PROGRAM POU_AxisClearError
VAR_INPUT
END_VAR
VAR
	fbAxis1Reset:MC_Reset;
	fbAxis2Reset:MC_Reset;
	fbAxis3Reset:MC_Reset;
	fbAxis4Reset:MC_Reset;
	fbAxis5Reset:MC_Reset;
	fbAxis6Reset:MC_Reset;
	
END_VAR

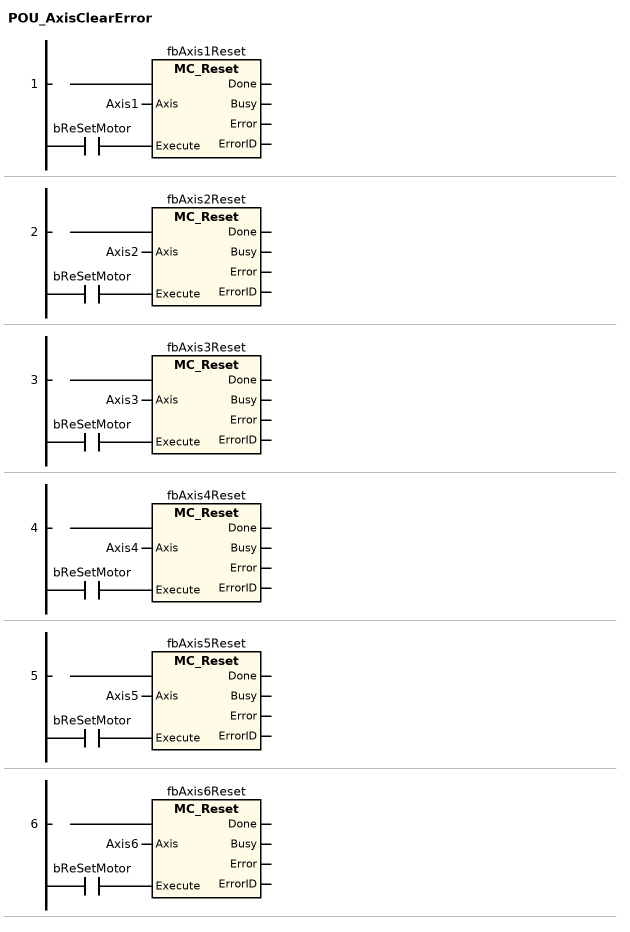
// NETWORK 1
fbAxis1Reset(Axis := Axis1, Execute := bReSetMotor); // MC_Reset

// NETWORK 2
fbAxis2Reset(Axis := Axis2, Execute := bReSetMotor); // MC_Reset

// NETWORK 3
fbAxis3Reset(Axis := Axis3, Execute := bReSetMotor); // MC_Reset

// NETWORK 4
fbAxis4Reset(Axis := Axis4, Execute := bReSetMotor); // MC_Reset

// NETWORK 5
fbAxis5Reset(Axis := Axis5, Execute := bReSetMotor); // MC_Reset

// NETWORK 6
fbAxis6Reset(Axis := Axis6, Execute := bReSetMotor); // MC_Reset

END_PROGRAM

(* stored: Version 1.1.0.1, ProductVersion 3.1.4022.18
   POU POU_AxisClearError: Id {af1272c6-fc94-4f03-a8f1-10ebb8289fc4}, SpecialFunc None *)
